FUNCTION_BLOCK DoorSensor (* Template for a simple Basic Function Block Type *)
  (* Standard: 61499-2 *)
  (* Version 1.0, 2019-05-09, jetbrains *)
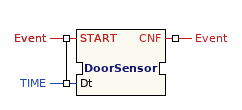
  EVENT_INPUT
    START WITH Dt; (* Normal Execution Request *)
    START; (* Normal Execution Request *)
  END_EVENT
  EVENT_OUTPUT
    CNF WITH doorOpen; (* Execution Confirmation *)
  END_EVENT
  VAR_INPUT
    Dt : TIME; (* Input event qualifier *)
  END_VAR
END_FUNCTION_BLOCK
